(* PLC project weighingscale, Dassault Systèmes ControlBuild 2024x *)
(* stored: creationDateTime 2023-10-04T11:03:51-01:00 *)

FUNCTION_BLOCK motion_lib.weighingscale
  VAR_OUTPUT
    Weight : INT := 0;
  END_VAR
  VAR
    status_act_prod : DINT := 0;
    m11 : REAL := 1.0;
    m12 : REAL := 0.0;
    m13 : REAL := 0.0;
    m14 : REAL := 0.0;
    m21 : REAL := 0.0;
    m22 : REAL := 1.0;
    m23 : REAL := 0.0;
    m24 : REAL := 0.0;
    m31 : REAL := 0.0;
    m32 : REAL := 0.0;
    m33 : REAL := 1.0;
    m34 : REAL := 0.0;
    m41 : REAL := 0.0;
    m42 : REAL := 0.0;
    m43 : REAL := 0.0;
    m44 : REAL := 1.0;
    weight : INT := 0;
  END_VAR

Weight := weight ;
weight := 0;
END_FUNCTION_BLOCK
